// TIA Portal V16 export
// export: Created 2024-05-13T12:47:21.62722Z, ExportSetting WithDefaults, DisplayName Totally Integrated Automation Portal, DisplayVersion V16 Update 6, DisplayName TIA Portal Version Control Interface, DisplayVersion V16 Update 2, DisplayName TIA Portal Openness, DisplayVersion V16 Update 6, DisplayName TIA Portal Test Suite Advanced, DisplayVersion V16, DisplayName SINAMICS Startdrive Advanced, DisplayVersion V16 Update 5, DisplayName SINAMICS Startdrive G130, G150, S120, S150, SINAMICS MV, S210, DisplayVersion V16 Update 5, DisplayName SINAMICS Startdrive G110M, G120, G120C, G120D, G120P, G115D, DisplayVersion V16 Update 5, DisplayName STEP 7 Professional, DisplayVersion V16 Update 6, DisplayName STEP 7 Safety, DisplayVersion V16, DisplayName WinCC Advanced, DisplayVersion V16 Update 6
FUNCTION_BLOCK "RH_OUT_2190TR"   // FB26, LAD
TITLE = Slat conveyor - 2190TR outputs
{ S7_Optimized_Access := 'TRUE' }
AUTHOR : JLA
VERSION : 0.1
// stored: AutoNumber true, IsIECCheckEnabled false, IsRetainMemResEnabled false, MemoryReserve 100, SetENOAutomatically false, UDAEnableTagReadback false
   VAR
      Diag { S7_SetPoint := 'True'} : "RMP_UDT_DIAG";   // Device diagnostics
      Status { S7_SetPoint := 'True'} : "RMP_UDT_DEV_STATUS";   // Device status information
      HMI_Status { S7_SetPoint := 'True'} : "RMP_HMI_DEV_STATUS";   // Device status information for HMI
      IO : Struct   // Device inputs and outputs
         Input : Struct
            Safety_switch : Bool;   // Safety switch
            Entry_pec : Bool;   // Entry photocell
            Exit_pec : Bool;   // Exit photocell
            Pulse_A : Bool;   // Pulse A
            Pulse_B : Bool;   // Pulse B
            Next_entry_pec : Bool;   // Next conveyor entry pec
            Prev_exit_pec : Bool;   // Previous conveyor exit pec
            Man_cnv_fwd : Bool;   // Forward
            Man_cnv_rev : Bool;   // Reverse
            Separation_pec : Bool;
            In_11 : Bool;
            In_12 : Bool;
            In_13 : Bool;
            In_14 : Bool;
            In_15 : Bool;
            In_16 : Bool;
            In_17 : Bool;
            In_18 : Bool;
            In_19 : Bool;
            In_20 : Bool;
            In_21 : Bool;
            In_22 : Bool;
            In_23 : Bool;
            In_24 : Bool;
            In_25 : Bool;
            In_26 : Bool;
            In_27 : Bool;
            In_28 : Bool;
            In_29 : Bool;
            In_30 : Bool;
            In_31 : Bool;
            In_32 : Bool;
         END_STRUCT;
         Output : Struct
            Out_1 : Bool;
            Out_2 : Bool;
            Out_3 : Bool;
            Out_4 : Bool;
            Out_5 : Bool;
            Out_6 : Bool;
            Out_7 : Bool;
            Out_8 : Bool;
            Out_9 : Bool;
            Out_10 : Bool;
            Out_11 : Bool;
            Out_12 : Bool;
            Out_13 : Bool;
            Out_14 : Bool;
            Out_15 : Bool;
            Out_16 : Bool;
            Out_17 : Bool;
            Out_18 : Bool;
            Out_19 : Bool;
            Out_20 : Bool;
            Out_21 : Bool;
            Out_22 : Bool;
            Out_23 : Bool;
            Out_24 : Bool;
            Out_25 : Bool;
            Out_26 : Bool;
            Out_27 : Bool;
            Out_28 : Bool;
            Out_29 : Bool;
            Out_30 : Bool;
            Out_31 : Bool;
            Out_32 : Bool;
         END_STRUCT;
      END_STRUCT;
      Flags : Struct   // Device auxilary flags
         Speed_1 : Bool;   // Speed selection 1
         Speed_2 : Bool;   // Speed selection 2
         Speed_3 : Bool;   // Speed selection 3
         Speed_4 : Bool;   // Speed selection 4
         Data_ok : Bool;   // Roll data present
         Entry_pec_fault : Bool;   // Entry pec fault
         Exit_pec_fault : Bool;   // Exit pec fault
         Buffering : Bool;   // Conveyor buffering rolls
         Separate_p : Bool;   // Exit pec neg pulse help bit
         Separate : Bool;   // Separate set reset help bit
         Device_stopped : Bool;
         Bit_11 : Bool;
         Bit_12 : Bool;
         Bit_13 : Bool;
         Bit_14 : Bool;
         Bit_15 : Bool;
         Bit_16 : Bool;
         Bit_17 : Bool;
         Bit_18 : Bool;
         Bit_19 : Bool;
         Bit_20 : Bool;
         Bit_21 : Bool;
         Bit_22 : Bool;
         Bit_23 : Bool;
         Bit_24 : Bool;
         Bit_25 : Bool;
         Bit_26 : Bool;
         Bit_27 : Bool;
         Bit_28 : Bool;
         Bit_29 : Bool;
         Bit_30 : Bool;
         Bit_31 : Bool;
         Bit_32 : Bool;
         Bit_33 : Bool;
         Bit_34 : Bool;
         Bit_35 : Bool;
         Bit_36 : Bool;
         Bit_37 : Bool;
         Bit_38 : Bool;
         Bit_39 : Bool;
         Bit_40 : Bool;
         Bit_41 : Bool;
         Bit_42 : Bool;
         Bit_43 : Bool;
         Bit_44 : Bool;
         Bit_45 : Bool;
         Bit_46 : Bool;
         Bit_47 : Bool;
         Bit_48 : Bool;
         Bit_49 : Bool;
         Bit_50 : Bool;
         Bit_51 : Bool;
         Bit_52 : Bool;
         Bit_53 : Bool;
         Bit_54 : Bool;
         Bit_55 : Bool;
         Bit_56 : Bool;
         Bit_57 : Bool;
         Bit_58 : Bool;
         Bit_59 : Bool;
         Bit_60 : Bool;
         Bit_61 : Bool;
         Bit_62 : Bool;
         Bit_63 : Bool;
      END_STRUCT;
      Data : Struct   // Device data
         Roll_width : Int;
         Position : Int;
         Target : Int;
         Data_int_4 : Int;
         Data_int_5 : Int;
         Data_int_6 : Int;
         Data_int_7 : Int;
         Data_int_8 : Int;
         Data_int_9 : Int;
         Data_int_10 : Int;
         Data_int_11 : Int;
         Data_int_12 : Int;
         Data_int_13 : Int;
         Data_int_14 : Int;
         Data_int_15 : Int;
         Data_int_16 : Int;
         Data_int_17 : Int;
         Data_int_18 : Int;
         Data_int_19 : Int;
         Data_int_20 : Int;
         Roll_front_end : DInt;
         Data_Dint_2 : DInt;
         Data_Dint_3 : DInt;
         Data_Dint_4 : DInt;
         Data_Dint_5 : DInt;
         Data_Dint_6 : DInt;
         Data_Dint_7 : DInt;
         Data_Dint_8 : DInt;
         Data_Dint_9 : DInt;
         Data_Dint_10 : DInt;
         Data_Dint_11 : DInt;
         Data_Dint_12 : DInt;
         Data_Dint_13 : DInt;
         Data_Dint_14 : DInt;
         Data_Dint_15 : DInt;
         Data_Dint_16 : DInt;
         Data_Dint_17 : DInt;
         HMI_alarms : Int;   // Alarms for KTP700
         Data_next : DWord;   // Conveyor data for next conveyor
         Data_prev : DWord;   // Conveyor data for previous conveyor
      END_STRUCT;
      Interlock { S7_SetPoint := 'True'} : "RMP_UDT_INTERLOCK";   // Device interlocks
      Control { S7_SetPoint := 'True'} : "RMP_UDT_CONTROL";   // Device control
      Frq { S7_SetPoint := 'True'} : "RMP_BIF_FRQ_SPD";   // Device frquency converter control
      Drive { S7_SetPoint := 'True'} : "RMP_FRQ_SPD";
      Encoder { S7_SetPoint := 'True'} : "RMP_BIF_CNV_ENC_CNT";
      Centering { S7_SetPoint := 'True'} : "RMP_BIF_CENTERING";
      Program_Alarm { S7_SetPoint := 'True'} : Array[1..16] of Program_Alarm;   // Device alarms
      Program_Event { S7_SetPoint := 'True'} : Array[1..8] of Program_Alarm;   // Device events
      Device_name { ExternalAccessible := 'False'; ExternalVisible := 'False'; ExternalWritable := 'False'} : String[30] := 'Slat conveyor - 865TR2190';
      RMP_PEC_FAULT_Instance_1 { S7_SetPoint := 'True'} : "RMP_PEC_FAULT";
      RMP_PEC_FAULT_Instance_2 { S7_SetPoint := 'True'} : "RMP_PEC_FAULT";
      RMP_ROLL_WIDTH_Instance { S7_SetPoint := 'True'} : "RMP_ROLL_WIDTH";
      RMP_CONV_DATA_Instance { ExternalAccessible := 'False'; ExternalVisible := 'False'; ExternalWritable := 'False'; S7_SetPoint := 'True'} : "RMP_CONV_DATA";
      RMP_SERV_COUNTER_Instance : "RMP_SERV_COUNTER";
      RMP_EMPTY_CNT_Instance { S7_SetPoint := 'True'} : "RMP_EMPTY_CNT";
      RMP_POSITIONING_Instance { S7_SetPoint := 'True'} : "RMP_POSITIONING";
      RMP_CNV_ENC_CNT_Instance { S7_SetPoint := 'True'} : "RMP_CNV_ENC_CNT";
      Event_1_delay { S7_SetPoint := 'True'} : TON_TIME;
      RMP_CNV_ENC_Instance { S7_SetPoint := 'True'} : "RMP_CNV_ENC";
      RMP_CENTERING_Instance { S7_SetPoint := 'True'} : "RMP_CENTERING";
      IEC_Timer_0_Instance { S7_SetPoint := 'True'} : TON_TIME;
      RMP_GAP_CONTROL_Instance { S7_SetPoint := 'True'} : "RMP_GAP_CONTROL";
      Entry_gap { S7_SetPoint := 'True'} : "RMP_BIF_GAP_CONTROL";
      ORG : Struct
         ORG_1 : Bool;
         ORG_2 : Bool;
         ORG_3 : Bool;
         ORG_4 : Bool;
         ORG_5 : Bool;
         ORG_6 : Bool;
         ORG_7 : Bool;
         ORG_8 : Bool;
      END_STRUCT;
      AUX : Struct
         Print_position : Bool;   // Calculate Printing position
         AUX_2 : Bool;
         AUX_3 : Bool;
         AUX_4 : Bool;
         AUX_5 : Bool;
         AUX_6 : Bool;
         AUX_7 : Bool;
         AUX_8 : Bool;
      END_STRUCT;
      RMP_SENSOR_DELAY_Instance { S7_SetPoint := 'True'} : "RMP_SENSOR_DELAY";
   END_VAR
   VAR_TEMP
      Temp_R : Real;
      Temp_I : Int;
      Temp_DI : DInt;
      Error : Bool;
      Error_number : Int;
      Replace : Struct
         Prev_rev : Bool;
         Next_fwd : Bool;
         Conveyor_data : Array[1..10] of DWord;
         Roll_width : Int;
      END_STRUCT;
      Error_nbr : Int;
      slow_speed : Int;
      seqStepNumber : Int;
      bTempCreepSpeed : Bool;   // Previous conveyor has rolldata
   END_VAR
   // // Interlock.Fwd : fwd interlocks
   // // Interlock.Fwd[1] : Safety switch open
   // // Interlock.Fwd[2] : Exit pec on and next is not running
   // // Interlock.Fwd[3] : Exit pec on and next is not ready
   // // Interlock.Fwd[4] : Rollers is not at down position
   // // Interlock.Fwd[5] : Belt is not at printer side
   // // Interlock.Fwd[6] : Roll at joint and prev is not running
   // // Interlock.Rev : rev interlocks
   // // Interlock.Rev[1] : Safety switch open
   // // Interlock.Rev[2] : Entry pec on and prev is not running
   // // Interlock.Rev[3] : Rollers is not at down position
   // // Interlock.Rev[4] : Entry pec on and prev is not ready
   // // Interlock.Rev[5] : Belt is not at printer side
   VAR_TEMP   // added for the SCL form of the ladder/FBD networks
      _w1 : Bool;
   END_VAR
BEGIN

REGION Network 1: Control area interface
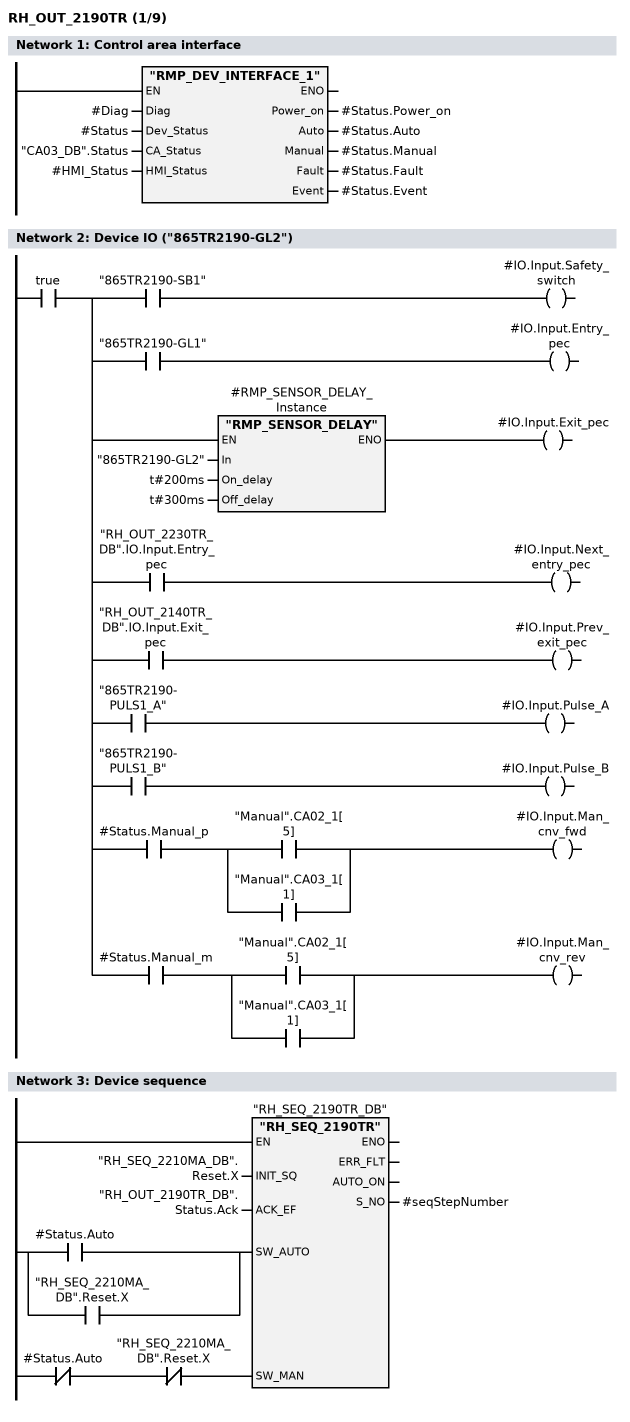
   RUNG wire#powerrail
      "RMP_DEV_INTERFACE_1"(Diag := #Diag, Dev_Status := #Status, CA_Status := "CA03_DB".Status, HMI_Status := #HMI_Status, Power_on => #Status.Power_on, Auto => #Status.Auto, Manual => #Status.Manual, Fault => #Status.Fault, Event => #Status.Event)
   END_RUNG
   // the same network as SCL:
   "RMP_DEV_INTERFACE_1"(Diag := #Diag,
                         Dev_Status := #Status,
                         CA_Status := "CA03_DB".Status,
                         HMI_Status := #HMI_Status,
                         Power_on => #Status.Power_on,
                         Auto => #Status.Auto,
                         Manual => #Status.Manual,
                         Fault => #Status.Fault,
                         Event => #Status.Event);
END_REGION

REGION Network 2: Device IO ("865TR2190-GL2")
   RUNG wire#powerrail
      Contact( true )
      wire#w1
      Contact( "865TR2190-SB1" )
      Coil( #IO.Input.Safety_switch )
   END_RUNG
   RUNG wire#w1
      Contact( "865TR2190-GL1" )
      Coil( #IO.Input.Entry_pec )
   END_RUNG
   RUNG wire#w1
      #RMP_SENSOR_DELAY_Instance(In := "865TR2190-GL2", On_delay := t#200ms, Off_delay := t#300ms)
      Coil( #IO.Input.Exit_pec )
   END_RUNG
   RUNG wire#w1
      Contact( "RH_OUT_2230TR_DB".IO.Input.Entry_pec )
      Coil( #IO.Input.Next_entry_pec )
   END_RUNG
   RUNG wire#w1
      Contact( "RH_OUT_2140TR_DB".IO.Input.Exit_pec )
      Coil( #IO.Input.Prev_exit_pec )
   END_RUNG
   RUNG wire#w1
      Contact( "865TR2190-PULS1_A" )
      Coil( #IO.Input.Pulse_A )
   END_RUNG
   RUNG wire#w1
      Contact( "865TR2190-PULS1_B" )
      Coil( #IO.Input.Pulse_B )
   END_RUNG
   RUNG wire#w1
      Contact( #Status.Manual_p )
      wire#w2
      Contact( "Manual".CA02_1[5] )
      wire#w3
      Coil( #IO.Input.Man_cnv_fwd )
   END_RUNG
   RUNG wire#w2
      Contact( "Manual".CA03_1[1] )
   END_RUNG wire#w3
   RUNG wire#w1
      Contact( #Status.Manual_m )
      wire#w4
      Contact( "Manual".CA02_1[5] )
      wire#w5
      Coil( #IO.Input.Man_cnv_rev )
   END_RUNG
   RUNG wire#w4
      Contact( "Manual".CA03_1[1] )
   END_RUNG wire#w5
   // the same network as SCL:
   #IO.Input.Safety_switch := true AND "865TR2190-SB1";
   #IO.Input.Entry_pec := true AND "865TR2190-GL1";
   #RMP_SENSOR_DELAY_Instance(EN := true,   // "RMP_SENSOR_DELAY"
                           In := "865TR2190-GL2",
                           On_delay := t#200ms,
                           Off_delay := t#300ms,
                           ENO => #_w1);
   #IO.Input.Exit_pec := #_w1;
   #IO.Input.Next_entry_pec := true AND "RH_OUT_2230TR_DB".IO.Input.Entry_pec;
   #IO.Input.Prev_exit_pec := true AND "RH_OUT_2140TR_DB".IO.Input.Exit_pec;
   #IO.Input.Pulse_A := true AND "865TR2190-PULS1_A";
   #IO.Input.Pulse_B := true AND "865TR2190-PULS1_B";
   #IO.Input.Man_cnv_fwd := true AND #Status.Manual_p AND ("Manual".CA02_1[5] OR "Manual".CA03_1[1]);
   #IO.Input.Man_cnv_rev := true AND #Status.Manual_m AND ("Manual".CA02_1[5] OR "Manual".CA03_1[1]);
END_REGION

REGION Network 3: Device sequence
   RUNG wire#powerrail
      "RH_SEQ_2190TR_DB"(SW_AUTO := wire#w1, SW_MAN := wire#w2, INIT_SQ := "RH_SEQ_2210MA_DB".Reset.X, ACK_EF := "RH_OUT_2190TR_DB".Status.Ack, ERR_FLT =>, AUTO_ON =>, S_NO => #seqStepNumber)
   END_RUNG
   RUNG wire#powerrail
      Contact( #Status.Auto )
   END_RUNG wire#w1
   RUNG wire#powerrail
      Contact( "RH_SEQ_2210MA_DB".Reset.X )
   END_RUNG wire#w1
   RUNG wire#powerrail
      I_Contact( #Status.Auto )
      I_Contact( "RH_SEQ_2210MA_DB".Reset.X )
   END_RUNG wire#w2
   // the same network as SCL:
   "RH_SEQ_2190TR_DB"(INIT_SQ := "RH_SEQ_2210MA_DB".Reset.X,   // "RH_SEQ_2190TR"
                      ACK_EF := "RH_OUT_2190TR_DB".Status.Ack,
                      SW_AUTO := #Status.Auto OR "RH_SEQ_2210MA_DB".Reset.X,
                      SW_MAN := NOT #Status.Auto AND NOT "RH_SEQ_2210MA_DB".Reset.X,
                      S_NO => #seqStepNumber);
END_REGION

REGION Network 4: Device stopped
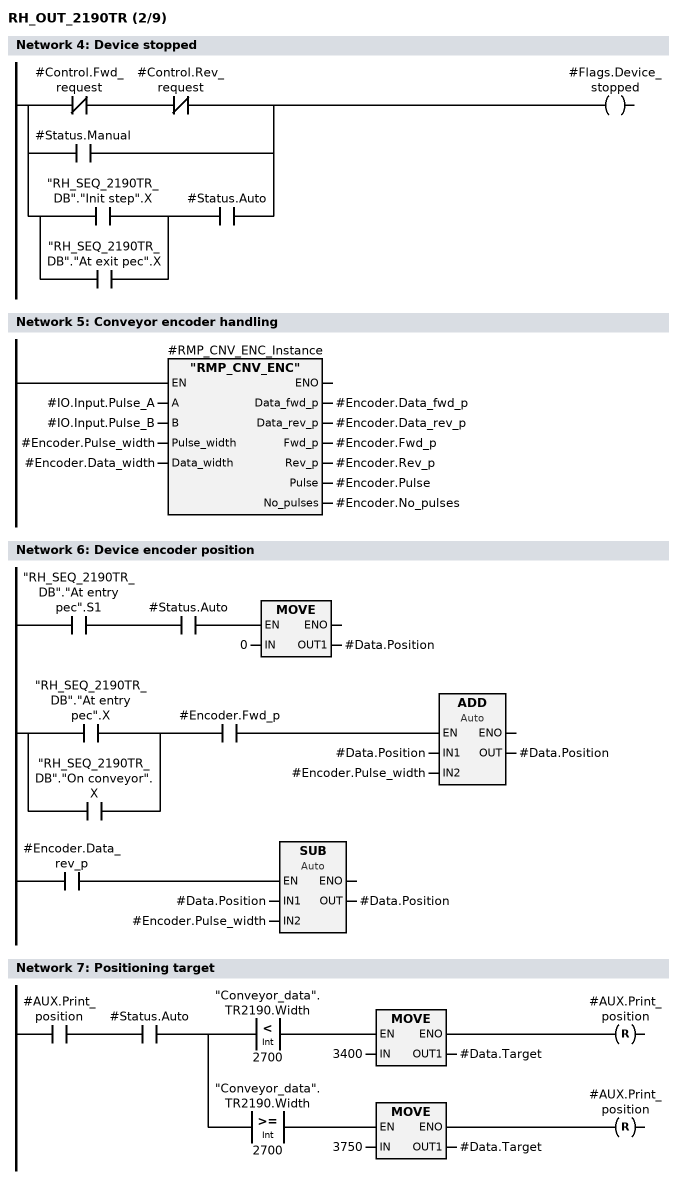
   RUNG wire#powerrail
      I_Contact( #Control.Fwd_request )
      I_Contact( #Control.Rev_request )
      wire#w1
      Coil( #Flags.Device_stopped )
   END_RUNG
   RUNG wire#powerrail
      Contact( #Status.Manual )
   END_RUNG wire#w1
   RUNG wire#powerrail
      Contact( "RH_SEQ_2190TR_DB"."Init step".X )
      wire#w2
      Contact( #Status.Auto )
   END_RUNG wire#w1
   RUNG wire#powerrail
      Contact( "RH_SEQ_2190TR_DB"."At exit pec".X )
   END_RUNG wire#w2
   // the same network as SCL:
   #Flags.Device_stopped := (NOT #Control.Fwd_request AND NOT #Control.Rev_request) OR #Status.Manual OR (("RH_SEQ_2190TR_DB"."Init step".X OR "RH_SEQ_2190TR_DB"."At exit pec".X) AND #Status.Auto);
END_REGION

REGION Network 5: Conveyor encoder handling
   RUNG wire#powerrail
      #RMP_CNV_ENC_Instance("A" := #IO.Input.Pulse_A, "B" := #IO.Input.Pulse_B, Pulse_width := #Encoder.Pulse_width, Data_width := #Encoder.Data_width, Data_fwd_p => #Encoder.Data_fwd_p, Data_rev_p => #Encoder.Data_rev_p, Fwd_p => #Encoder.Fwd_p, Rev_p => #Encoder.Rev_p, Pulse => #Encoder.Pulse, No_pulses => #Encoder.No_pulses)
   END_RUNG
   // the same network as SCL:
   #RMP_CNV_ENC_Instance("A" := #IO.Input.Pulse_A,   // "RMP_CNV_ENC"
                         "B" := #IO.Input.Pulse_B,
                         Pulse_width := #Encoder.Pulse_width,
                         Data_width := #Encoder.Data_width,
                         Data_fwd_p => #Encoder.Data_fwd_p,
                         Data_rev_p => #Encoder.Data_rev_p,
                         Fwd_p => #Encoder.Fwd_p,
                         Rev_p => #Encoder.Rev_p,
                         Pulse => #Encoder.Pulse,
                         No_pulses => #Encoder.No_pulses);
END_REGION

REGION Network 6: Device encoder position
   RUNG wire#powerrail
      Contact( "RH_SEQ_2190TR_DB"."At entry pec".S1 )
      Contact( #Status.Auto )
      Move(in := 0, out1 => #Data.Position)
   END_RUNG
   RUNG wire#powerrail
      Contact( "RH_SEQ_2190TR_DB"."At entry pec".X )
      wire#w1
      Contact( #Encoder.Fwd_p )
      Add(in1 := #Data.Position, in2 := #Encoder.Pulse_width, out => #Data.Position)
   END_RUNG
   RUNG wire#powerrail
      Contact( "RH_SEQ_2190TR_DB"."On conveyor".X )
   END_RUNG wire#w1
   RUNG wire#powerrail
      Contact( #Encoder.Data_rev_p )
      Sub(in1 := #Data.Position, in2 := #Encoder.Pulse_width, out => #Data.Position)
   END_RUNG
   // the same network as SCL:
   IF "RH_SEQ_2190TR_DB"."At entry pec".S1 AND #Status.Auto THEN #Data.Position := 0; END_IF;
   IF ("RH_SEQ_2190TR_DB"."At entry pec".X OR "RH_SEQ_2190TR_DB"."On conveyor".X) AND #Encoder.Fwd_p THEN
       #Data.Position := #Data.Position + #Encoder.Pulse_width;
   END_IF;
   IF #Encoder.Data_rev_p THEN #Data.Position := #Data.Position - #Encoder.Pulse_width; END_IF;
END_REGION

REGION Network 7: Positioning target
   RUNG wire#powerrail
      Contact( #AUX.Print_position )
      Contact( #Status.Auto )
      wire#w1
      { S7_Templates := "SrcType := Int" } LT_Contact(in1 := "Conveyor_data".TR2190.Width, in2 := 2700)
      Move(in := 3400, out1 => #Data.Target)
      R_Coil( #AUX.Print_position )
   END_RUNG
   RUNG wire#w1
      { S7_Templates := "SrcType := Int" } GE_Contact(in1 := "Conveyor_data".TR2190.Width, in2 := 2700)
      Move(in := 3750, out1 => #Data.Target)
      R_Coil( #AUX.Print_position )
   END_RUNG
   // the same network as SCL:
   #_w1 := #AUX.Print_position AND #Status.Auto;
   IF #_w1 AND ("Conveyor_data".TR2190.Width < 2700) THEN
       #Data.Target := 3400;
       #AUX.Print_position := FALSE;
   END_IF;
   IF #_w1 AND ("Conveyor_data".TR2190.Width >= 2700) THEN
       #Data.Target := 3750;
       #AUX.Print_position := FALSE;
   END_IF;
END_REGION

REGION Network 8: Service counter
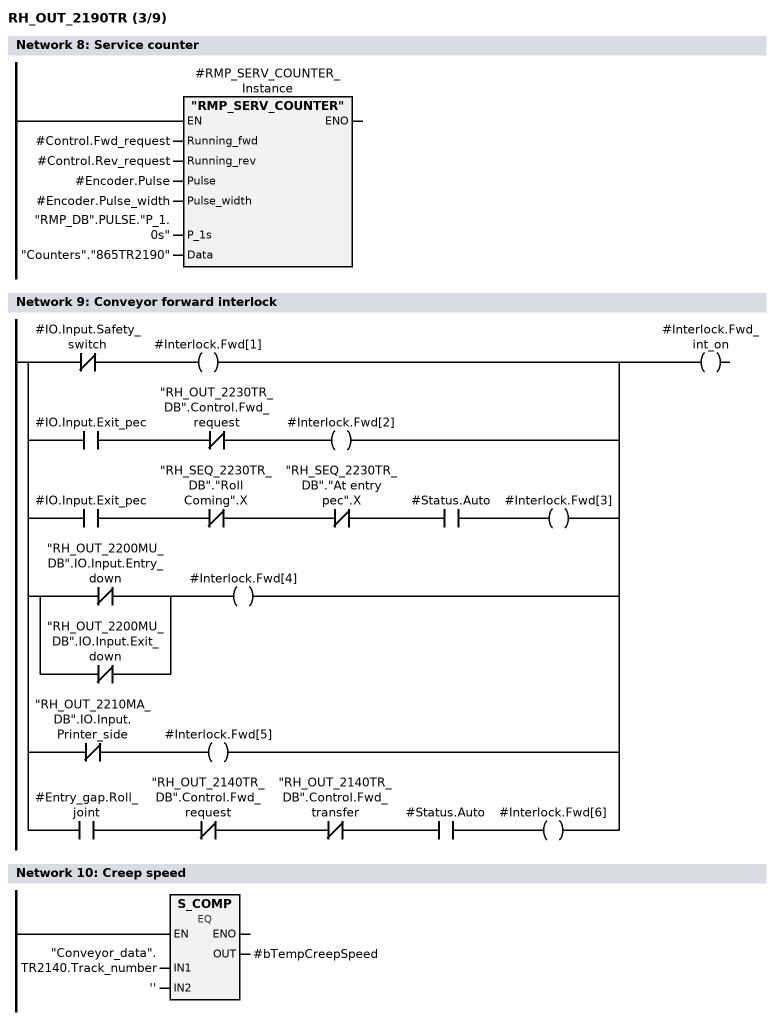
   RUNG wire#powerrail
      #RMP_SERV_COUNTER_Instance(Running_fwd := #Control.Fwd_request, Running_rev := #Control.Rev_request, Pulse := #Encoder.Pulse, Pulse_width := #Encoder.Pulse_width, P_1s := "RMP_DB".PULSE."P_1.0s", Data := "Counters"."865TR2190")
   END_RUNG
   // the same network as SCL:
   #RMP_SERV_COUNTER_Instance(Running_fwd := #Control.Fwd_request,   // "RMP_SERV_COUNTER"
                           Running_rev := #Control.Rev_request,
                           Pulse := #Encoder.Pulse,
                           Pulse_width := #Encoder.Pulse_width,
                           P_1s := "RMP_DB".PULSE."P_1.0s",
                           Data := "Counters"."865TR2190");
END_REGION

REGION Network 9: Conveyor forward interlock
   RUNG wire#powerrail
      I_Contact( #IO.Input.Safety_switch )
      Coil( #Interlock.Fwd[1] )
      wire#w1
      Coil( #Interlock.Fwd_int_on )
   END_RUNG
   RUNG wire#powerrail
      Contact( #IO.Input.Exit_pec )
      I_Contact( "RH_OUT_2230TR_DB".Control.Fwd_request )
      Coil( #Interlock.Fwd[2] )
   END_RUNG wire#w1
   RUNG wire#powerrail
      Contact( #IO.Input.Exit_pec )
      I_Contact( "RH_SEQ_2230TR_DB"."Roll Coming".X )
      I_Contact( "RH_SEQ_2230TR_DB"."At entry pec".X )
      Contact( #Status.Auto )
      Coil( #Interlock.Fwd[3] )
   END_RUNG wire#w1
   RUNG wire#powerrail
      I_Contact( "RH_OUT_2200MU_DB".IO.Input.Entry_down )
      wire#w2
      Coil( #Interlock.Fwd[4] )
   END_RUNG wire#w1
   RUNG wire#powerrail
      I_Contact( "RH_OUT_2200MU_DB".IO.Input.Exit_down )
   END_RUNG wire#w2
   RUNG wire#powerrail
      I_Contact( "RH_OUT_2210MA_DB".IO.Input.Printer_side )
      Coil( #Interlock.Fwd[5] )
   END_RUNG wire#w1
   RUNG wire#powerrail
      Contact( #Entry_gap.Roll_joint )
      I_Contact( "RH_OUT_2140TR_DB".Control.Fwd_request )
      I_Contact( "RH_OUT_2140TR_DB".Control.Fwd_transfer )
      Contact( #Status.Auto )
      Coil( #Interlock.Fwd[6] )
   END_RUNG wire#w1
   // the same network as SCL:
   #Interlock.Fwd[1] := NOT #IO.Input.Safety_switch;
   #Interlock.Fwd[2] := #IO.Input.Exit_pec AND NOT "RH_OUT_2230TR_DB".Control.Fwd_request;
   #Interlock.Fwd[3] := #IO.Input.Exit_pec AND NOT "RH_SEQ_2230TR_DB"."Roll Coming".X AND NOT "RH_SEQ_2230TR_DB"."At entry pec".X AND #Status.Auto;
   #Interlock.Fwd[4] := NOT "RH_OUT_2200MU_DB".IO.Input.Entry_down OR NOT "RH_OUT_2200MU_DB".IO.Input.Exit_down;
   #Interlock.Fwd[5] := NOT "RH_OUT_2210MA_DB".IO.Input.Printer_side;
   #Interlock.Fwd[6] := #Entry_gap.Roll_joint AND NOT "RH_OUT_2140TR_DB".Control.Fwd_request AND NOT "RH_OUT_2140TR_DB".Control.Fwd_transfer AND #Status.Auto;
   #Interlock.Fwd_int_on := NOT #IO.Input.Safety_switch OR (#IO.Input.Exit_pec AND NOT "RH_OUT_2230TR_DB".Control.Fwd_request) OR (#IO.Input.Exit_pec AND NOT "RH_SEQ_2230TR_DB"."Roll Coming".X AND NOT "RH_SEQ_2230TR_DB"."At entry pec".X AND #Status.Auto) OR NOT "RH_OUT_2200MU_DB".IO.Input.Entry_down OR NOT "RH_OUT_2200MU_DB".IO.Input.Exit_down OR NOT "RH_OUT_2210MA_DB".IO.Input.Printer_side OR (#Entry_gap.Roll_joint AND NOT "RH_OUT_2140TR_DB".Control.Fwd_request AND NOT "RH_OUT_2140TR_DB".Control.Fwd_transfer AND #Status.Auto);
END_REGION

REGION Network 10: Creep speed
   RUNG wire#powerrail
      { S7_Templates := "[relation := EQ, src_type := String]" } S_COMP(IN1 := "Conveyor_data".TR2140.Track_number, IN2 := '', OUT => #bTempCreepSpeed)
   END_RUNG
   // the same network as SCL:
   S_COMP(IN1 := "Conveyor_data".TR2140.Track_number, IN2 := '', OUT => #bTempCreepSpeed);
END_REGION

REGION Network 11: Conveyor forward
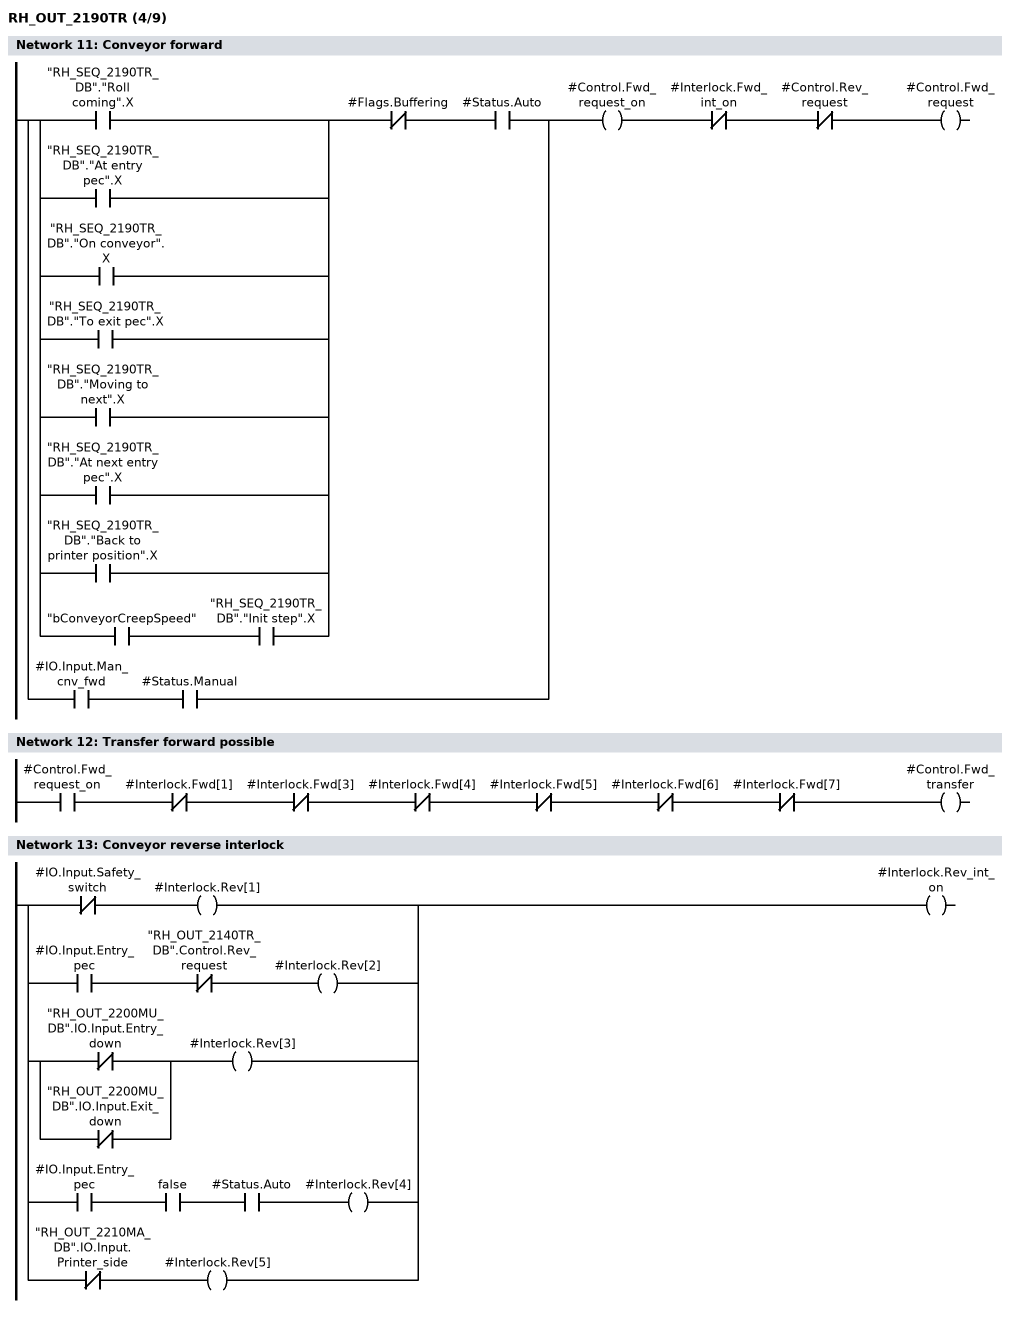
   RUNG wire#powerrail
      Contact( "RH_SEQ_2190TR_DB"."Roll coming".X )
      wire#w1
      I_Contact( #Flags.Buffering )
      Contact( #Status.Auto )
      wire#w2
      Coil( #Control.Fwd_request_on )
      I_Contact( #Interlock.Fwd_int_on )
      I_Contact( #Control.Rev_request )
      Coil( #Control.Fwd_request )
   END_RUNG
   RUNG wire#powerrail
      Contact( "RH_SEQ_2190TR_DB"."At entry pec".X )
   END_RUNG wire#w1
   RUNG wire#powerrail
      Contact( "RH_SEQ_2190TR_DB"."On conveyor".X )
   END_RUNG wire#w1
   RUNG wire#powerrail
      Contact( "RH_SEQ_2190TR_DB"."To exit pec".X )
   END_RUNG wire#w1
   RUNG wire#powerrail
      Contact( "RH_SEQ_2190TR_DB"."Moving to next".X )
   END_RUNG wire#w1
   RUNG wire#powerrail
      Contact( "RH_SEQ_2190TR_DB"."At next entry pec".X )
   END_RUNG wire#w1
   RUNG wire#powerrail
      Contact( "RH_SEQ_2190TR_DB"."Back to printer position".X )
   END_RUNG wire#w1
   RUNG wire#powerrail
      Contact( "bConveyorCreepSpeed" )
      Contact( "RH_SEQ_2190TR_DB"."Init step".X )
   END_RUNG wire#w1
   RUNG wire#powerrail
      Contact( #IO.Input.Man_cnv_fwd )
      Contact( #Status.Manual )
   END_RUNG wire#w2
   // the same network as SCL:
   #Control.Fwd_request_on := (("RH_SEQ_2190TR_DB"."Roll coming".X OR "RH_SEQ_2190TR_DB"."At entry pec".X OR "RH_SEQ_2190TR_DB"."On conveyor".X OR "RH_SEQ_2190TR_DB"."To exit pec".X OR "RH_SEQ_2190TR_DB"."Moving to next".X OR "RH_SEQ_2190TR_DB"."At next entry pec".X OR "RH_SEQ_2190TR_DB"."Back to printer position".X OR ("bConveyorCreepSpeed" AND "RH_SEQ_2190TR_DB"."Init step".X)) AND NOT #Flags.Buffering AND #Status.Auto) OR (#IO.Input.Man_cnv_fwd AND #Status.Manual);
   #Control.Fwd_request := #Control.Fwd_request_on AND NOT #Interlock.Fwd_int_on AND NOT #Control.Rev_request;
END_REGION

REGION Network 12: Transfer forward possible
   RUNG wire#powerrail
      Contact( #Control.Fwd_request_on )
      I_Contact( #Interlock.Fwd[1] )
      I_Contact( #Interlock.Fwd[3] )
      I_Contact( #Interlock.Fwd[4] )
      I_Contact( #Interlock.Fwd[5] )
      I_Contact( #Interlock.Fwd[6] )
      I_Contact( #Interlock.Fwd[7] )
      Coil( #Control.Fwd_transfer )
   END_RUNG
   // the same network as SCL:
   #Control.Fwd_transfer := #Control.Fwd_request_on AND NOT #Interlock.Fwd[1] AND NOT #Interlock.Fwd[3] AND NOT #Interlock.Fwd[4] AND NOT #Interlock.Fwd[5] AND NOT #Interlock.Fwd[6] AND NOT #Interlock.Fwd[7];
END_REGION

REGION Network 13: Conveyor reverse interlock
   RUNG wire#powerrail
      I_Contact( #IO.Input.Safety_switch )
      Coil( #Interlock.Rev[1] )
      wire#w1
      Coil( #Interlock.Rev_int_on )
   END_RUNG
   RUNG wire#powerrail
      Contact( #IO.Input.Entry_pec )
      I_Contact( "RH_OUT_2140TR_DB".Control.Rev_request )
      Coil( #Interlock.Rev[2] )
   END_RUNG wire#w1
   RUNG wire#powerrail
      I_Contact( "RH_OUT_2200MU_DB".IO.Input.Entry_down )
      wire#w2
      Coil( #Interlock.Rev[3] )
   END_RUNG wire#w1
   RUNG wire#powerrail
      I_Contact( "RH_OUT_2200MU_DB".IO.Input.Exit_down )
   END_RUNG wire#w2
   RUNG wire#powerrail
      Contact( #IO.Input.Entry_pec )
      Contact( false )
      Contact( #Status.Auto )
      Coil( #Interlock.Rev[4] )
   END_RUNG wire#w1
   RUNG wire#powerrail
      I_Contact( "RH_OUT_2210MA_DB".IO.Input.Printer_side )
      Coil( #Interlock.Rev[5] )
   END_RUNG wire#w1
   // the same network as SCL:
   #Interlock.Rev[1] := NOT #IO.Input.Safety_switch;
   #Interlock.Rev[2] := #IO.Input.Entry_pec AND NOT "RH_OUT_2140TR_DB".Control.Rev_request;
   #Interlock.Rev[3] := NOT "RH_OUT_2200MU_DB".IO.Input.Entry_down OR NOT "RH_OUT_2200MU_DB".IO.Input.Exit_down;
   #Interlock.Rev[4] := #IO.Input.Entry_pec AND false AND #Status.Auto;
   #Interlock.Rev[5] := NOT "RH_OUT_2210MA_DB".IO.Input.Printer_side;
   #Interlock.Rev_int_on := NOT #IO.Input.Safety_switch OR (#IO.Input.Entry_pec AND NOT "RH_OUT_2140TR_DB".Control.Rev_request) OR NOT "RH_OUT_2200MU_DB".IO.Input.Entry_down OR NOT "RH_OUT_2200MU_DB".IO.Input.Exit_down OR (#IO.Input.Entry_pec AND false AND #Status.Auto) OR NOT "RH_OUT_2210MA_DB".IO.Input.Printer_side;
END_REGION

REGION Network 14: Conveyor reverse
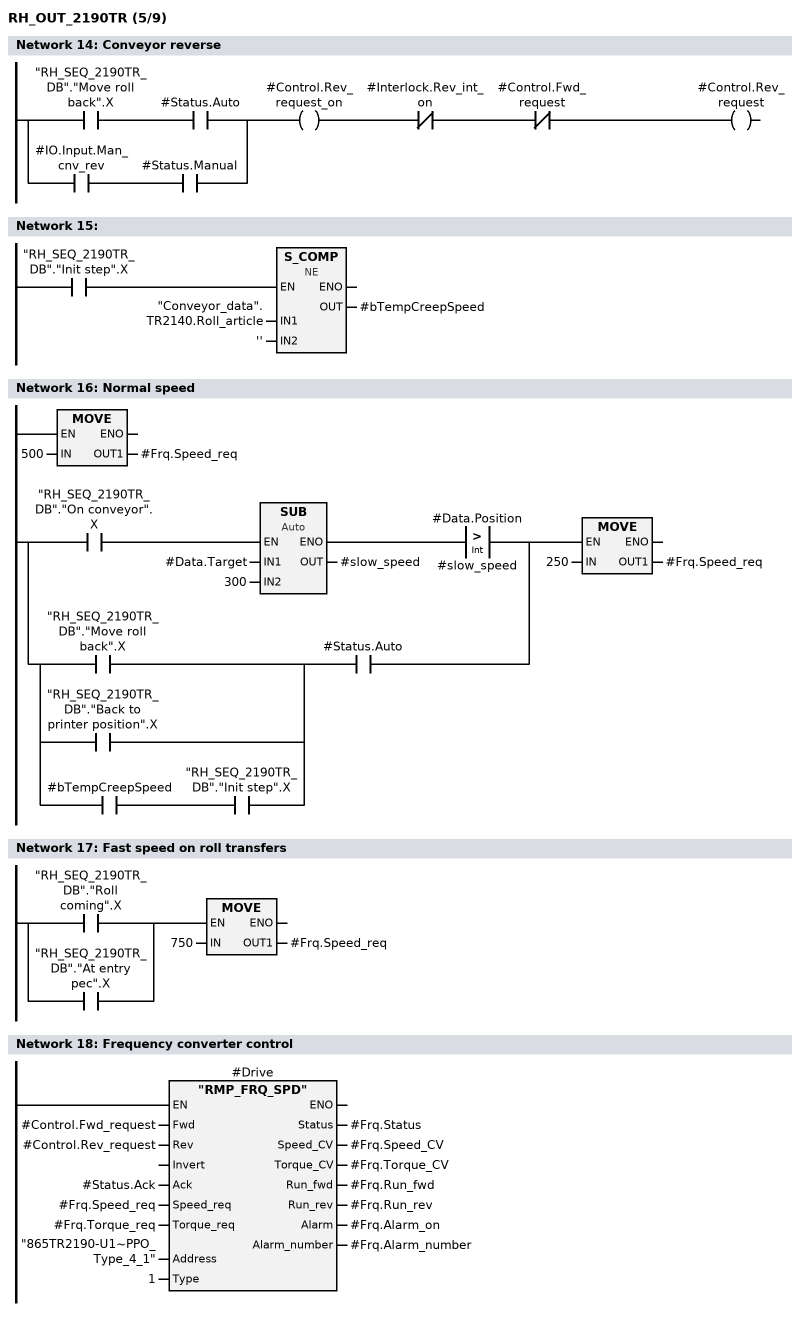
   RUNG wire#powerrail
      Contact( "RH_SEQ_2190TR_DB"."Move roll back".X )
      Contact( #Status.Auto )
      wire#w1
      Coil( #Control.Rev_request_on )
      I_Contact( #Interlock.Rev_int_on )
      I_Contact( #Control.Fwd_request )
      Coil( #Control.Rev_request )
   END_RUNG
   RUNG wire#powerrail
      Contact( #IO.Input.Man_cnv_rev )
      Contact( #Status.Manual )
   END_RUNG wire#w1
   // the same network as SCL:
   #Control.Rev_request_on := ("RH_SEQ_2190TR_DB"."Move roll back".X AND #Status.Auto) OR (#IO.Input.Man_cnv_rev AND #Status.Manual);
   #Control.Rev_request := #Control.Rev_request_on AND NOT #Interlock.Rev_int_on AND NOT #Control.Fwd_request;
END_REGION

REGION Network 15
   RUNG wire#powerrail
      Contact( "RH_SEQ_2190TR_DB"."Init step".X )
      { S7_Templates := "[relation := NE, src_type := String]" } S_COMP(IN1 := "Conveyor_data".TR2140.Roll_article, IN2 := '', OUT => #bTempCreepSpeed)
   END_RUNG
   // the same network as SCL:
   IF "RH_SEQ_2190TR_DB"."Init step".X THEN
       S_COMP(IN1 := "Conveyor_data".TR2140.Roll_article, IN2 := '', OUT => #bTempCreepSpeed);
   END_IF;
END_REGION

REGION Network 16: Normal speed
   RUNG wire#powerrail
      { S7_GenerateENO := "TRUE" } Move(in := 500, out1 => #Frq.Speed_req)
   END_RUNG
   RUNG wire#powerrail
      Contact( "RH_SEQ_2190TR_DB"."On conveyor".X )
      Sub(in1 := #Data.Target, in2 := 300, out => #slow_speed)
      { S7_Templates := "SrcType := Int" } GT_Contact(in1 := #Data.Position, in2 := #slow_speed)
      wire#w1
      { S7_GenerateENO := "TRUE" } Move(in := 250, out1 => #Frq.Speed_req)
   END_RUNG
   RUNG wire#powerrail
      Contact( "RH_SEQ_2190TR_DB"."Move roll back".X )
      wire#w2
      Contact( #Status.Auto )
   END_RUNG wire#w1
   RUNG wire#powerrail
      Contact( "RH_SEQ_2190TR_DB"."Back to printer position".X )
   END_RUNG wire#w2
   RUNG wire#powerrail
      Contact( #bTempCreepSpeed )
      Contact( "RH_SEQ_2190TR_DB"."Init step".X )
   END_RUNG wire#w2
   // the same network as SCL:
   #Frq.Speed_req := 500;
   IF "RH_SEQ_2190TR_DB"."On conveyor".X THEN #slow_speed := #Data.Target - 300; END_IF;
   IF ("RH_SEQ_2190TR_DB"."On conveyor".X AND (#Data.Position > #slow_speed)) OR (("RH_SEQ_2190TR_DB"."Move roll back".X OR "RH_SEQ_2190TR_DB"."Back to printer position".X OR (#bTempCreepSpeed AND "RH_SEQ_2190TR_DB"."Init step".X)) AND #Status.Auto) THEN
       #Frq.Speed_req := 250;
   END_IF;
END_REGION

REGION Network 17: Fast speed on roll transfers
   RUNG wire#powerrail
      Contact( "RH_SEQ_2190TR_DB"."Roll coming".X )
      wire#w1
      { S7_GenerateENO := "TRUE" } Move(in := 750, out1 => #Frq.Speed_req)
   END_RUNG
   RUNG wire#powerrail
      Contact( "RH_SEQ_2190TR_DB"."At entry pec".X )
   END_RUNG wire#w1
   // the same network as SCL:
   IF "RH_SEQ_2190TR_DB"."Roll coming".X OR "RH_SEQ_2190TR_DB"."At entry pec".X THEN
       #Frq.Speed_req := 750;
   END_IF;
END_REGION

REGION Network 18: Frequency converter control
   RUNG wire#powerrail
      #Drive(Fwd := #Control.Fwd_request, Rev := #Control.Rev_request, Invert :=, Ack := #Status.Ack, Speed_req := #Frq.Speed_req, Torque_req := #Frq.Torque_req, Address := "865TR2190-U1~PPO_Type_4_1", "Type" := 1, Status => #Frq.Status, Speed_CV => #Frq.Speed_CV, Torque_CV => #Frq.Torque_CV, Run_fwd => #Frq.Run_fwd, Run_rev => #Frq.Run_rev, Alarm => #Frq.Alarm_on, Alarm_number => #Frq.Alarm_number)
   END_RUNG
   // the same network as SCL:
   #Drive(Fwd := #Control.Fwd_request,   // "RMP_FRQ_SPD"
          Rev := #Control.Rev_request,
          Ack := #Status.Ack,
          Speed_req := #Frq.Speed_req,
          Torque_req := #Frq.Torque_req,
          Address := "865TR2190-U1~PPO_Type_4_1",
          "Type" := 1,
          Status => #Frq.Status,
          Speed_CV => #Frq.Speed_CV,
          Torque_CV => #Frq.Torque_CV,
          Run_fwd => #Frq.Run_fwd,
          Run_rev => #Frq.Run_rev,
          Alarm => #Frq.Alarm_on,
          Alarm_number => #Frq.Alarm_number);
END_REGION

REGION Network 19: Roll centering on conveyor
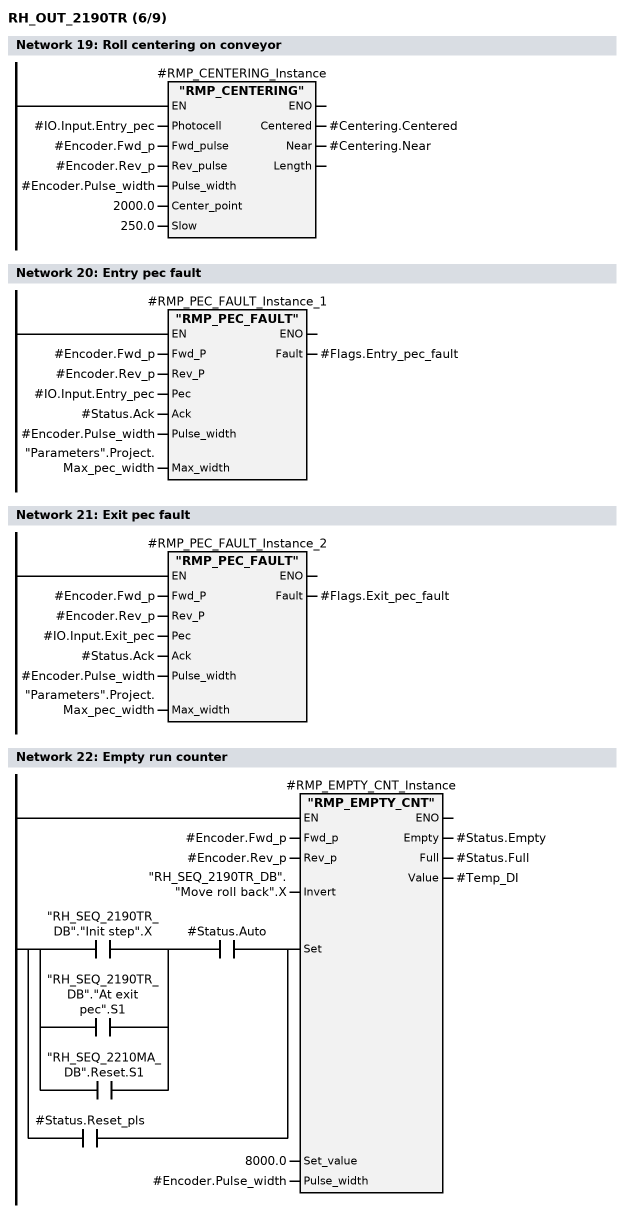
   RUNG wire#powerrail
      #RMP_CENTERING_Instance(Photocell := #IO.Input.Entry_pec, Fwd_pulse := #Encoder.Fwd_p, Rev_pulse := #Encoder.Rev_p, Pulse_width := #Encoder.Pulse_width, Center_point := 2000.0, Slow := 250.0, Centered => #Centering.Centered, Near => #Centering.Near, Length =>)
   END_RUNG
   // the same network as SCL:
   #RMP_CENTERING_Instance(Photocell := #IO.Input.Entry_pec,   // "RMP_CENTERING"
                           Fwd_pulse := #Encoder.Fwd_p,
                           Rev_pulse := #Encoder.Rev_p,
                           Pulse_width := #Encoder.Pulse_width,
                           Center_point := 2000.0,
                           Slow := 250.0,
                           Centered => #Centering.Centered,
                           Near => #Centering.Near);
END_REGION

REGION Network 20: Entry pec fault
   RUNG wire#powerrail
      #RMP_PEC_FAULT_Instance_1(Fwd_P := #Encoder.Fwd_p, Rev_P := #Encoder.Rev_p, Pec := #IO.Input.Entry_pec, Ack := #Status.Ack, Pulse_width := #Encoder.Pulse_width, Max_width := "Parameters".Project.Max_pec_width, Fault => #Flags.Entry_pec_fault)
   END_RUNG
   // the same network as SCL:
   #RMP_PEC_FAULT_Instance_1(Fwd_P := #Encoder.Fwd_p,   // "RMP_PEC_FAULT"
                           Rev_P := #Encoder.Rev_p,
                           Pec := #IO.Input.Entry_pec,
                           Ack := #Status.Ack,
                           Pulse_width := #Encoder.Pulse_width,
                           Max_width := "Parameters".Project.Max_pec_width,
                           Fault => #Flags.Entry_pec_fault);
END_REGION

REGION Network 21: Exit pec fault
   RUNG wire#powerrail
      #RMP_PEC_FAULT_Instance_2(Fwd_P := #Encoder.Fwd_p, Rev_P := #Encoder.Rev_p, Pec := #IO.Input.Exit_pec, Ack := #Status.Ack, Pulse_width := #Encoder.Pulse_width, Max_width := "Parameters".Project.Max_pec_width, Fault => #Flags.Exit_pec_fault)
   END_RUNG
   // the same network as SCL:
   #RMP_PEC_FAULT_Instance_2(Fwd_P := #Encoder.Fwd_p,   // "RMP_PEC_FAULT"
                           Rev_P := #Encoder.Rev_p,
                           Pec := #IO.Input.Exit_pec,
                           Ack := #Status.Ack,
                           Pulse_width := #Encoder.Pulse_width,
                           Max_width := "Parameters".Project.Max_pec_width,
                           Fault => #Flags.Exit_pec_fault);
END_REGION

REGION Network 22: Empty run counter
   RUNG wire#powerrail
      #RMP_EMPTY_CNT_Instance(Set := wire#w2, Fwd_p := #Encoder.Fwd_p, Rev_p := #Encoder.Rev_p, Invert := "RH_SEQ_2190TR_DB"."Move roll back".X, Set_value := 8000.0, Pulse_width := #Encoder.Pulse_width, Empty => #Status.Empty, Full => #Status.Full, Value => #Temp_DI)
   END_RUNG
   RUNG wire#powerrail
      Contact( "RH_SEQ_2190TR_DB"."Init step".X )
      wire#w1
      Contact( #Status.Auto )
   END_RUNG wire#w2
   RUNG wire#powerrail
      Contact( "RH_SEQ_2190TR_DB"."At exit pec".S1 )
   END_RUNG wire#w1
   RUNG wire#powerrail
      Contact( "RH_SEQ_2210MA_DB".Reset.S1 )
   END_RUNG wire#w1
   RUNG wire#powerrail
      Contact( #Status.Reset_pls )
   END_RUNG wire#w2
   // the same network as SCL:
   #RMP_EMPTY_CNT_Instance(Fwd_p := #Encoder.Fwd_p,   // "RMP_EMPTY_CNT"
                           Rev_p := #Encoder.Rev_p,
                           Invert := "RH_SEQ_2190TR_DB"."Move roll back".X,
                           Set := (("RH_SEQ_2190TR_DB"."Init step".X OR "RH_SEQ_2190TR_DB"."At exit pec".S1 OR "RH_SEQ_2210MA_DB".Reset.S1) AND #Status.Auto) OR #Status.Reset_pls,
                           Set_value := 8000.0,
                           Pulse_width := #Encoder.Pulse_width,
                           Empty => #Status.Empty,
                           Full => #Status.Full,
                           Value => #Temp_DI);
END_REGION

REGION Network 23: Gap control
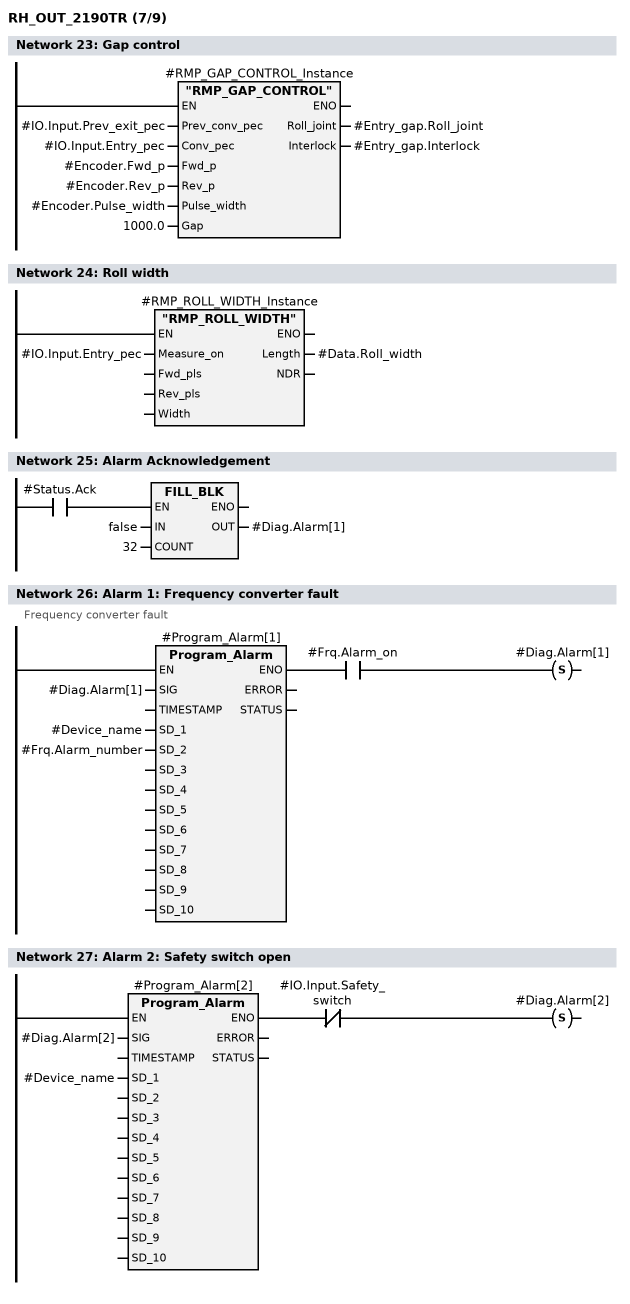
   RUNG wire#powerrail
      #RMP_GAP_CONTROL_Instance(Prev_conv_pec := #IO.Input.Prev_exit_pec, Conv_pec := #IO.Input.Entry_pec, Fwd_p := #Encoder.Fwd_p, Rev_p := #Encoder.Rev_p, Pulse_width := #Encoder.Pulse_width, Gap := 1000.0, Roll_joint => #Entry_gap.Roll_joint, Interlock => #Entry_gap.Interlock)
   END_RUNG
   // the same network as SCL:
   #RMP_GAP_CONTROL_Instance(Prev_conv_pec := #IO.Input.Prev_exit_pec,   // "RMP_GAP_CONTROL"
                           Conv_pec := #IO.Input.Entry_pec,
                           Fwd_p := #Encoder.Fwd_p,
                           Rev_p := #Encoder.Rev_p,
                           Pulse_width := #Encoder.Pulse_width,
                           Gap := 1000.0,
                           Roll_joint => #Entry_gap.Roll_joint,
                           Interlock => #Entry_gap.Interlock);
END_REGION

REGION Network 24: Roll width
   RUNG wire#powerrail
      #RMP_ROLL_WIDTH_Instance(Measure_on := #IO.Input.Entry_pec, Fwd_pls :=, Rev_pls :=, Width :=, Length => #Data.Roll_width, NDR =>)
   END_RUNG
   // the same network as SCL:
   #RMP_ROLL_WIDTH_Instance(Measure_on := #IO.Input.Entry_pec, Length => #Data.Roll_width);   // "RMP_ROLL_WIDTH"
END_REGION

REGION Network 25: Alarm Acknowledgement
   RUNG wire#powerrail
      Contact( #Status.Ack )
      FillBlockI(in := false, count := 32, out => #Diag.Alarm[1])
   END_RUNG
   // the same network as SCL:
   IF #Status.Ack THEN FILL_BLK(IN := false, COUNT := 32, OUT => #Diag.Alarm[1]); END_IF;
END_REGION

REGION Network 26: Alarm 1: Frequency converter fault
   // Frequency converter fault
   RUNG wire#powerrail
      #Program_Alarm[1].Program_Alarm(SIG := #Diag.Alarm[1], TIMESTAMP :=, SD_1 := #Device_name, SD_2 := #Frq.Alarm_number, SD_3 :=, SD_4 :=, SD_5 :=, SD_6 :=, SD_7 :=, SD_8 :=, SD_9 :=, SD_10 :=, Error =>, Status =>)
      Contact( #Frq.Alarm_on )
      S_Coil( #Diag.Alarm[1] )
   END_RUNG
   // the same network as SCL:
   #Program_Alarm[1](SIG := #Diag.Alarm[1], SD_1 := #Device_name, SD_2 := #Frq.Alarm_number, ENO => #_w1);   // Program_Alarm
   IF #_w1 AND #Frq.Alarm_on THEN #Diag.Alarm[1] := TRUE; END_IF;
END_REGION

REGION Network 27: Alarm 2: Safety switch open
   RUNG wire#powerrail
      #Program_Alarm[2].Program_Alarm(SIG := #Diag.Alarm[2], TIMESTAMP :=, SD_1 := #Device_name, SD_2 :=, SD_3 :=, SD_4 :=, SD_5 :=, SD_6 :=, SD_7 :=, SD_8 :=, SD_9 :=, SD_10 :=, Error =>, Status =>)
      I_Contact( #IO.Input.Safety_switch )
      S_Coil( #Diag.Alarm[2] )
   END_RUNG
   // the same network as SCL:
   #Program_Alarm[2](SIG := #Diag.Alarm[2], SD_1 := #Device_name, ENO => #_w1);   // Program_Alarm
   IF #_w1 AND NOT #IO.Input.Safety_switch THEN #Diag.Alarm[2] := TRUE; END_IF;
END_REGION

REGION Network 28: Alarm 3: Entry photocell fault
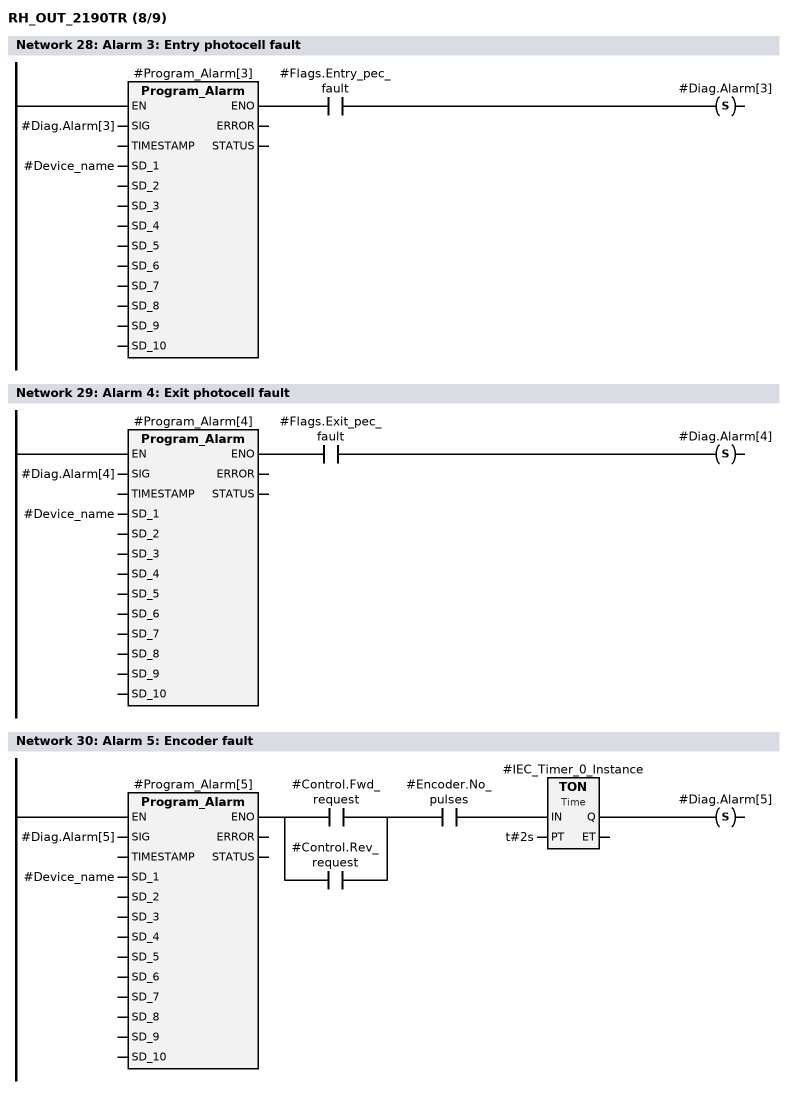
   RUNG wire#powerrail
      #Program_Alarm[3].Program_Alarm(SIG := #Diag.Alarm[3], TIMESTAMP :=, SD_1 := #Device_name, SD_2 :=, SD_3 :=, SD_4 :=, SD_5 :=, SD_6 :=, SD_7 :=, SD_8 :=, SD_9 :=, SD_10 :=, Error =>, Status =>)
      Contact( #Flags.Entry_pec_fault )
      S_Coil( #Diag.Alarm[3] )
   END_RUNG
   // the same network as SCL:
   #Program_Alarm[3](SIG := #Diag.Alarm[3], SD_1 := #Device_name, ENO => #_w1);   // Program_Alarm
   IF #_w1 AND #Flags.Entry_pec_fault THEN #Diag.Alarm[3] := TRUE; END_IF;
END_REGION

REGION Network 29: Alarm 4: Exit photocell fault
   RUNG wire#powerrail
      #Program_Alarm[4].Program_Alarm(SIG := #Diag.Alarm[4], TIMESTAMP :=, SD_1 := #Device_name, SD_2 :=, SD_3 :=, SD_4 :=, SD_5 :=, SD_6 :=, SD_7 :=, SD_8 :=, SD_9 :=, SD_10 :=, Error =>, Status =>)
      Contact( #Flags.Exit_pec_fault )
      S_Coil( #Diag.Alarm[4] )
   END_RUNG
   // the same network as SCL:
   #Program_Alarm[4](SIG := #Diag.Alarm[4], SD_1 := #Device_name, ENO => #_w1);   // Program_Alarm
   IF #_w1 AND #Flags.Exit_pec_fault THEN #Diag.Alarm[4] := TRUE; END_IF;
END_REGION

REGION Network 30: Alarm 5: Encoder fault
   RUNG wire#powerrail
      #Program_Alarm[5].Program_Alarm(SIG := #Diag.Alarm[5], TIMESTAMP :=, SD_1 := #Device_name, SD_2 :=, SD_3 :=, SD_4 :=, SD_5 :=, SD_6 :=, SD_7 :=, SD_8 :=, SD_9 :=, SD_10 :=, Error =>, Status =>)
      wire#w1
      Contact( #Control.Fwd_request )
      wire#w2
      Contact( #Encoder.No_pulses )
      { S7_Templates := "time_type := Time" } #IEC_Timer_0_Instance.TON(pt := t#2s, et =>)
      S_Coil( #Diag.Alarm[5] )
   END_RUNG
   RUNG wire#w1
      Contact( #Control.Rev_request )
   END_RUNG wire#w2
   // the same network as SCL:
   #Program_Alarm[5](SIG := #Diag.Alarm[5], SD_1 := #Device_name, ENO => #_w1);   // Program_Alarm
   #IEC_Timer_0_Instance(IN := #_w1 AND (#Control.Fwd_request OR #Control.Rev_request) AND #Encoder.No_pulses,   // TON
                         PT := t#2s);
   IF #IEC_Timer_0_Instance.Q THEN #Diag.Alarm[5] := TRUE; END_IF;
END_REGION

REGION Network 31: Alarm 6: Frequency converter safety fault
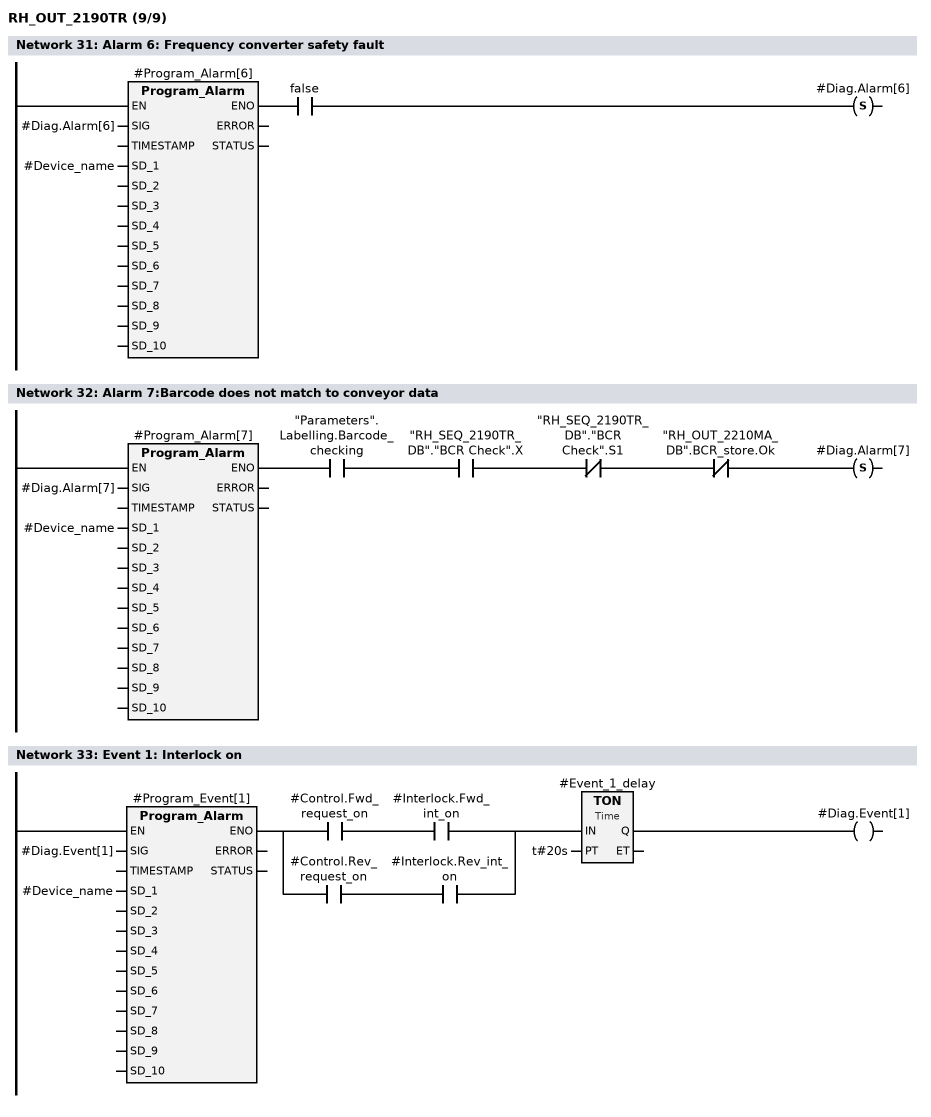
   RUNG wire#powerrail
      #Program_Alarm[6].Program_Alarm(SIG := #Diag.Alarm[6], TIMESTAMP :=, SD_1 := #Device_name, SD_2 :=, SD_3 :=, SD_4 :=, SD_5 :=, SD_6 :=, SD_7 :=, SD_8 :=, SD_9 :=, SD_10 :=, Error =>, Status =>)
      Contact( false )
      S_Coil( #Diag.Alarm[6] )
   END_RUNG
   // the same network as SCL:
   #Program_Alarm[6](SIG := #Diag.Alarm[6], SD_1 := #Device_name, ENO => #_w1);   // Program_Alarm
   IF #_w1 AND false THEN #Diag.Alarm[6] := TRUE; END_IF;
END_REGION

REGION Network 32: Alarm 7:Barcode does not match to conveyor data
   RUNG wire#powerrail
      #Program_Alarm[7].Program_Alarm(SIG := #Diag.Alarm[7], TIMESTAMP :=, SD_1 := #Device_name, SD_2 :=, SD_3 :=, SD_4 :=, SD_5 :=, SD_6 :=, SD_7 :=, SD_8 :=, SD_9 :=, SD_10 :=, Error =>, Status =>)
      Contact( "Parameters".Labelling.Barcode_checking )
      Contact( "RH_SEQ_2190TR_DB"."BCR Check".X )
      I_Contact( "RH_SEQ_2190TR_DB"."BCR Check".S1 )
      I_Contact( "RH_OUT_2210MA_DB".BCR_store.Ok )
      S_Coil( #Diag.Alarm[7] )
   END_RUNG
   // the same network as SCL:
   #Program_Alarm[7](SIG := #Diag.Alarm[7], SD_1 := #Device_name, ENO => #_w1);   // Program_Alarm
   IF #_w1 AND "Parameters".Labelling.Barcode_checking AND "RH_SEQ_2190TR_DB"."BCR Check".X AND NOT "RH_SEQ_2190TR_DB"."BCR Check".S1 AND NOT "RH_OUT_2210MA_DB".BCR_store.Ok THEN
       #Diag.Alarm[7] := TRUE;
   END_IF;
END_REGION

REGION Network 33: Event 1: Interlock on
   RUNG wire#powerrail
      #Program_Event[1].Program_Alarm(SIG := #Diag.Event[1], TIMESTAMP :=, SD_1 := #Device_name, SD_2 :=, SD_3 :=, SD_4 :=, SD_5 :=, SD_6 :=, SD_7 :=, SD_8 :=, SD_9 :=, SD_10 :=, Error =>, Status =>)
      wire#w1
      Contact( #Control.Fwd_request_on )
      Contact( #Interlock.Fwd_int_on )
      wire#w2
      { S7_Templates := "time_type := Time" } #Event_1_delay.TON(pt := t#20s, et =>)
      Coil( #Diag.Event[1] )
   END_RUNG
   RUNG wire#w1
      Contact( #Control.Rev_request_on )
      Contact( #Interlock.Rev_int_on )
   END_RUNG wire#w2
   // the same network as SCL:
   #Program_Event[1](SIG := #Diag.Event[1], SD_1 := #Device_name, ENO => #_w1);   // Program_Alarm
   #Event_1_delay(IN := #_w1 AND ((#Control.Fwd_request_on AND #Interlock.Fwd_int_on) OR (#Control.Rev_request_on AND #Interlock.Rev_int_on)),   // TON
                  PT := t#20s);
   #Diag.Event[1] := #Event_1_delay.Q;
END_REGION
END_FUNCTION_BLOCK
